PROGRAM XV03_DiagnosticsHelper
VAR
END_VAR

METHOD Parse : REFERENCE TO FB_XV03_DiagnosticsParser

VAR_INST
	fbXV03DiagnosisOptions	: FB_XV03_DiagnosticsParser;
END_VAR
Parse REF= fbXV03DiagnosisOptions;
END_METHOD

END_PROGRAM

(* stored: Version 1.1.0.1, ProductVersion 3.1.4024.13
   POU XV03_DiagnosticsHelper: Id {118e4d92-a0c8-0e86-12ea-136dc8c90737}, SpecialFunc None
   Method Parse: Id {7ebb7a8b-688e-05ee-3fdb-a499c0352b0f} *)
